FUNCTION_BLOCK FB_CleaningProcessStateProduction EXTENDS FB_CleaningProcessStateBase
VAR_INPUT
END_VAR
VAR_OUTPUT
END_VAR
VAR
END_VAR

METHOD mCleaningOp : BOOL
VAR_INPUT
	sI_Operation : EN_CLEANING_OP;
END_VAR
//Switch to production mode if no operation active
IF I_MachineStatus.pSafetyOk AND I_MachineStatus.pMachineReady AND NOT bL_DevOpActive THEN
  IF sI_Operation = eOPCAPENTER THEN
    I_ParentCallback.mChangeState(EN_Cleaning_State.Capping);
  ELSIF sI_Operation = eOPCAPEXIT THEN
    I_ParentCallback.mChangeState(EN_Cleaning_State.CappingExit);
  ELSIF sI_Operation = eOPCLEAN THEN
    I_ParentCallback.mChangeState(EN_Cleaning_State.Cleaning);
  ELSIF sI_Operation = eOPPURGE THEN
    I_ParentCallback.mChangeState(EN_Cleaning_State.Capping);
  END_IF
END_IF
END_METHOD

METHOD mDevOpDone : BOOL
VAR_INPUT
END_VAR
;//HOA TEST commented: no wait position with pneumatic axis I_ParentCallback.mChangeState(EN_Cleaning_State.Wait);
END_METHOD

METHOD mEntryAction
VAR_INPUT
END_VAR
iL_CurrentStep := 0;

// Launch initial command to bring system to production mode
bL_DevOpActive := I_ParentCallback.mSetMode(EN_CLEANING_OP.eOPGOTOPROD);
END_METHOD

METHOD mProduction : BOOL
VAR_INPUT
END_VAR
//Request production mode - implement in SubClass
mProduction := TRUE;
END_METHOD

METHOD mService : BOOL
VAR_INPUT
END_VAR
//Switch to service mode
IF NOT bL_DevOpActive THEN
	I_ParentCallback.mChangeState(EN_Cleaning_State.Service);
END_IF
END_METHOD

METHOD mStateAction
VAR_INPUT
END_VAR

VAR
	sL_DeviceStatus: ST_CLEANING_DEV_STATUS;
END_VAR
sL_DeviceStatus := I_ParentCallback.pDeviceStatus;

//If not MachineReady go to wait mode
(*HOA TEST commented
IF I_MachineStatus.pSafetyOk AND NOT bL_DevOpActive THEN
	IF NOT I_MachineStatus.pMachineReady THEN
		bL_DevOpActive := I_ParentCallback.mSetMode(EN_CLEANING_OP.eOPGOTOWAIT);
	END_IF
END_IF
*)
IF bL_DevOpActive THEN
	mDevOp();	
END_IF

//If error go to error mode
IF sL_DeviceStatus.bError THEN
	I_ParentCallback.mChangeState(EN_Cleaning_State.Error);
END_IF

SUPER^.pInitDone := TRUE;
END_METHOD

END_FUNCTION_BLOCK

(* stored: Version 1.1.0.1, ProductVersion 3.1.4024.11
   POU FB_CleaningProcessStateProduction: Id {20fc1865-5267-4568-8f97-a317031cd5ca}, SpecialFunc None
   Method mCleaningOp: Id {f540ad56-c850-4585-915a-7d676d8f40c3}
   Method mDevOpDone: Id {2703c9c0-045b-46db-aea5-556da8ceb618}
   Method mEntryAction: Id {19d481d5-380e-43fd-9eae-03ac829b17f4}
   Method mProduction: Id {4b363e8f-0bbd-4c6f-b1b2-b2de1e51bd77}
   Method mService: Id {9b549eea-b1db-419b-bfd9-ad4fcbda2e57}
   Method mStateAction: Id {b282738e-fdfc-40ca-9147-df9c83cd23ad} *)
